// TIA Portal V20 export
// export: Created 2026-04-20T18:50:18.2379397Z, ExportSetting WithDefaults, DisplayName Totally Integrated Automation Portal, DisplayVersion V20, DisplayName TIA Portal Openness, DisplayVersion V20, DisplayName TIA Portal Version Control Interface, DisplayVersion V20, DisplayName STEP 7 Professional, DisplayVersion V20, DisplayName STEP 7 Safety, DisplayVersion V20, DisplayName WinCC Basic/Comfort/Advanced, DisplayVersion V20
TYPE "UDT_EquipmentModule"
// stored: IsFailsafeCompliant false
   STRUCT
      moduleId : Int := 0;   // Unique module identifier within the unit
      moduleName : String[32] := 'Module';   // Human-readable module name
      moduleType : SInt := 1;   // Function: 1=Dosing 2=Heating 3=Stirring 4=Draining
      valves { S7_SetPoint := 'True'} : Array[1..4] of "UDT_ControlValve";   // Control valves belonging to this module
   END_STRUCT;
END_TYPE
